(* CoDeSys 2.3.9.50 project: 2E.pr6 *)
(* Libraries: STANDARD.LB6 5.6.98 12:03:02 *)

(* POU MAIN, LD *)
PROGRAM MAIN
VAR
	A AT %IX0.0: BOOL;
	B AT %IX0.1: BOOL;
	C AT %IX0.2: BOOL;
	Buzzer AT %QX0.0: BOOL;
	LightB AT %QX0.1: BOOL;
	LightC AT %QX0.2: BOOL;
	LightA AT %QX0.3: BOOL;
	Reset AT %IX0.7: BOOL;
END_VAR
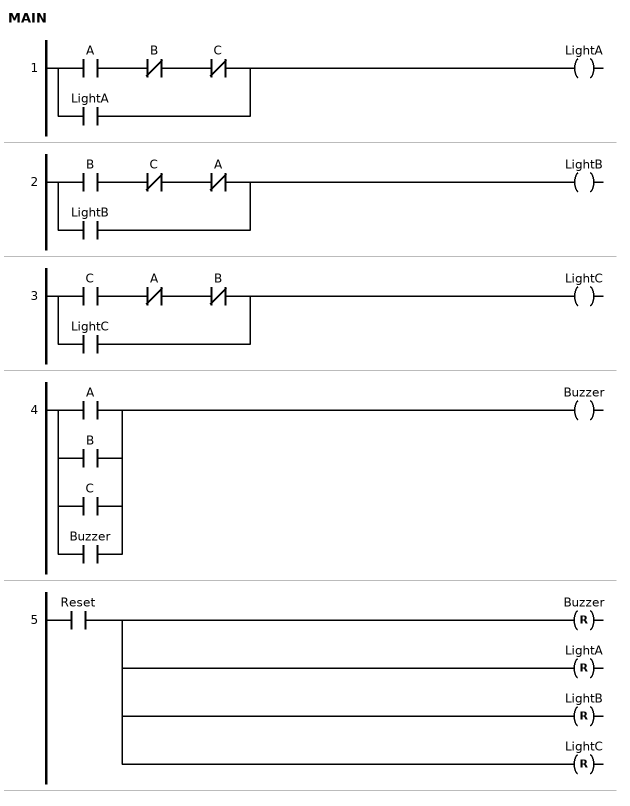
_LD_ (* Ladder Diagram *)
NETWORK 1
	{ [A] - [/B] - [/C] | [LightA] } --- (LightA)
NETWORK 2
	{ [B] - [/C] - [/A] | [LightB] } --- (LightB)
NETWORK 3
	{ [C] - [/A] - [/B] | [LightC] } --- (LightC)
NETWORK 4
	{ [A] | [B] | [C] | [Buzzer] } --- (Buzzer)
NETWORK 5
	[Reset] --- (R Buzzer) (R LightA) (R LightB) (R LightC)
_END_LD_
(* the same logic as Structured Text *)
(* Network 1 *)
LightA := A AND NOT B AND NOT C OR LightA;
(* Network 2 *)
LightB := B AND NOT C AND NOT A OR LightB;
(* Network 3 *)
LightC := C AND NOT A AND NOT B OR LightC;
(* Network 4 *)
Buzzer := A OR B OR C OR Buzzer;
(* Network 5 *)
IF Reset THEN Buzzer := FALSE; LightA := FALSE; LightB := FALSE; LightC := FALSE; END_IF;
END_PROGRAM

(* Visualisation Q2E
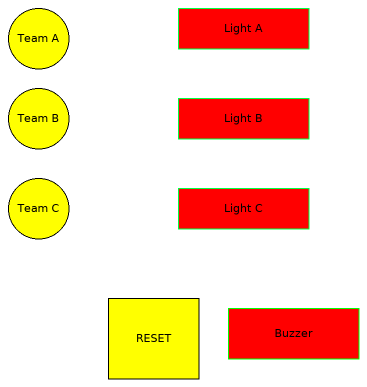
ellipse at (80,30)-(141,91): text "Team A"; alarm colour if %IX0.0; toggles %IX0.0
ellipse at (80,110)-(141,171): text "Team B"; alarm colour if %IX0.1; toggles %IX0.1
ellipse at (80,200)-(141,261): text "Team C"; alarm colour if %IX0.2; toggles %IX0.2
rectangle at (250,30)-(381,71): text "Light A"; alarm colour if %QX0.3
rectangle at (250,210)-(381,251): text "Light C"; alarm colour if %QX0.2
rectangle at (250,120)-(381,161): text "Light B"; alarm colour if %QX0.1
rounded rectangle at (180,320)-(271,401): text "RESET"; alarm colour if %IX0.7; toggles %IX0.7
rectangle at (300,330)-(431,381): text "Buzzer"; alarm colour if %QX0.0
*)
